# EPICS autosave request: ipApp/Db/SR570preamp_settings.req
#FILE... SR570preamp_settings.req
#USAGE... SR570.db fields autosave'd.
$(P)$(A)bias_put.VAL
$(P)$(A)bias_tweak.VAL
$(P)$(A)bias_on.VAL
$(P)$(A)off_u_put.VAL
$(P)$(A)offset_u_tweak.VAL
$(P)$(A)offset_cal.VAL
$(P)$(A)filter_type.VAL
$(P)$(A)low_freq.VAL
$(P)$(A)high_freq.VAL
$(P)$(A)offset_on.VAL
$(P)$(A)offset_sign.VAL
$(P)$(A)offset_num.VAL
$(P)$(A)offset_unit.VAL
$(P)$(A)gain_mode.VAL
$(P)$(A)invert_on.VAL
$(P)$(A)blank_on.VAL
$(P)$(A)sens_num.VAL
$(P)$(A)sens_unit.VAL
